// TIA Portal project "cyclic_interrupt" (V18)

(* hardware
DEVICE "S7-1200 station_1"  S7-1200 Station
   slot 0: "Rack_0"  S7-1200 Rack  Rack  V1.0
   slot 1: "PLC_1"  CPU 1214C DC/DC/DC  6ES7 214-1AG40-0XB0  V4.6
*)

// ===== PLC "PLC_1"  CPU 1214C DC/DC/DC =====

VAR_GLOBAL   // PLC tag table "Default tag table"
   "Tag_1" AT %Q0.0 : Bool;
   "Tag_2" AT %MW0 : Int;
   "Tag_3" AT %I0.0 : Bool;
   "Tag_4" AT %I0.1 : Bool;
   "Tag_5" AT %MW2 : Int;
   "Tag_6" AT %MD4 : UDInt;
   "Tag_7" AT %MD8 : UDInt;
   "Tag_8" AT %MW10 : Word;
END_VAR

ORGANIZATION_BLOCK "Main"   // OB1, LAD, ProgramCycle
TITLE = "Main Program Sweep (Cycle)"
{ S7_Optimized_Access := 'TRUE' }
VERSION : 0.1
// cet_cint
   VAR_INPUT
      Initial_Call : Bool;   // Initial call of this OB
      Remanence : Bool;   // =True, if remanent data are available
   END_VAR
BEGIN

REGION Network 1
   // cycle 1ms değerindedir
   // bu örnekte 1 sn oldu
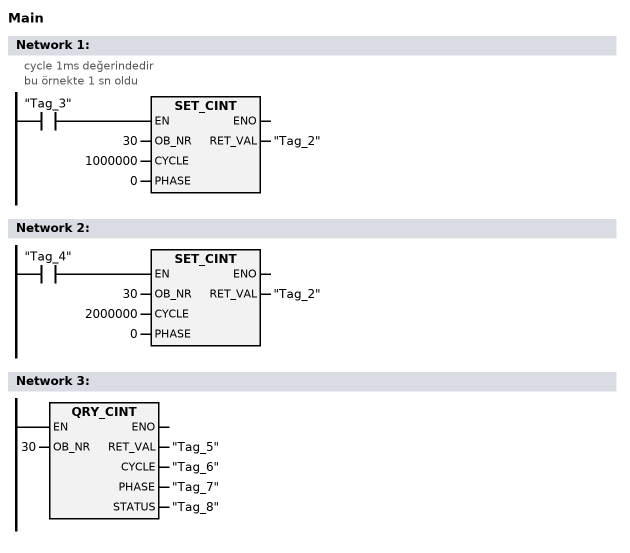
   IF "Tag_3" THEN "Tag_2" := SET_CINT(OB_NR := 30, CYCLE := 1000000, PHASE := 0); END_IF;
END_REGION

REGION Network 2
   IF "Tag_4" THEN "Tag_2" := SET_CINT(OB_NR := 30, CYCLE := 2000000, PHASE := 0); END_IF;
END_REGION

REGION Network 3
   "Tag_5" := QRY_CINT(OB_NR := 30, CYCLE => "Tag_6", PHASE => "Tag_7", STATUS => "Tag_8");
END_REGION
END_ORGANIZATION_BLOCK

ORGANIZATION_BLOCK "Cyclic interrupt"   // OB30, LAD, CyclicInterrupt
{ S7_Optimized_Access := 'TRUE' }
VERSION : 0.1
   VAR_INPUT
      Initial_Call : Bool;   // Initial call of this OB
      Event_Count : Int;   // Events discarded
   END_VAR
BEGIN

REGION Network 1
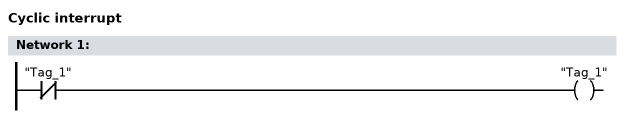
   RUNG wire#powerrail
      I_Contact( "Tag_1" )
      Coil( "Tag_1" )
   END_RUNG
   // the same network as SCL:
   "Tag_1" := NOT "Tag_1";
END_REGION
END_ORGANIZATION_BLOCK